// TIA Portal V21 export
TYPE "lubricationSystemIOs"
   STRUCT
      self { ExternalAccessible := 'False'; ExternalVisible := 'False'; ExternalWritable := 'False'} : "lubricationSystemInterface";
      localModeSwitch : "LBC_typeDigitalSignalInterface";
      btnStart : "LBC_typeDigitalSignalInterface";
      btnStop : "LBC_typeDigitalSignalInterface";
      btnReset : "LBC_typeDigitalSignalInterface";
      oilPump1SelSwitch : "LBC_typeDigitalSignalInterface";
      oilPump2SelSwitch : "LBC_typeDigitalSignalInterface";
      oilPreparationSwitch : "LBC_typeDigitalSignalInterface";
      returnOilFlowSwitch : "LBC_typeDigitalSignalInterface";
      oilLevelMax : "LBC_typeDigitalSignalInterface";
      oilLevelMid : "LBC_typeDigitalSignalInterface";
      oilLevelMin : "LBC_typeDigitalSignalInterface";
      oilTempSwitchHigh : "LBC_typeDigitalSignalInterface";   // TRUE - temp ok
      oilTempSwitchLow : "LBC_typeDigitalSignalInterface";
      fbPump1 : "LBC_typeDigitalSignalInterface";
      fbPump2 : "LBC_typeDigitalSignalInterface";
      pump1Fault : "LBC_typeDigitalSignalInterface";
      pump2Fault : "LBC_typeDigitalSignalInterface";
      oilTempTank : "LBC_typeAnalogInputInterface";
      oilPump1 : "LBC_typeMotorStarterInterface";
      oilPump2 : "LBC_typeMotorStarterInterface";
      returnOilTemp : "LBC_typeAnalogInputInterface";
      oilFlow : "LBC_typeAnalogInputInterface";
      inletWaterTemperature : "LBC_typeAnalogInputInterface";
      outletWaterTemperature : "LBC_typeAnalogInputInterface";
      inletOilTemperature : "LBC_typeAnalogInputInterface";
      inletOilPressure : "LBC_typeAnalogInputInterface";
      pump1Start : "LBC_typeDigitalSignalInterface";
      pump2Start : "LBC_typeDigitalSignalInterface";
      heaterOn : "LBC_typeDigitalSignalInterface";
      waterVlvOpen : "LBC_typeDigitalSignalInterface";
      oilToCoolerVlv : "LBC_typeDigitalSignalInterface";
   END_STRUCT;
END_TYPE
